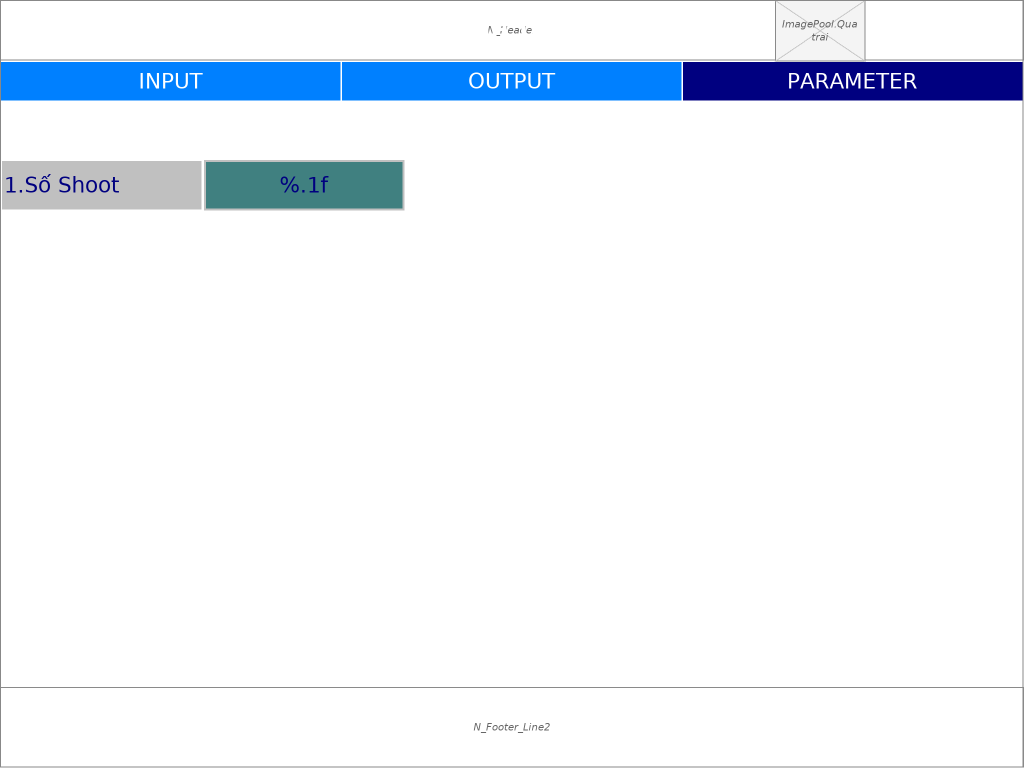
VISUALIZATION N_Parameter_2  // 1024x768
    Frame (0,0 1024x60)
        shows N_Header()
    Rectangle (0,61 341x40), "INPUT"
        OnMouseClick: change screen: N_PLC_I2
    Rectangle (341,61 341x40), "OUTPUT"
        OnMouseClick: change screen: N_PLC_O2
    Rectangle (682,61 341x40), "PARAMETER"
        OnMouseClick: change screen: N_Parameter_2
    Textfield (363,5 400x50), "MÀN HÌNH THÔNG SỐ TRẠM 2"
    Rectangle (1,160 201x50), "1.Số Shoot"
    Textfield (204,160 200x50), "%.1f", text variable: nShoot2
    Image (775,0 90x61), image: ImagePool.Qua trai
        OnMouseClick: change screen: N_Parameter_1
    Frame (0,687 1024x80)
        shows N_Footer_Line2()
END_VISUALIZATION

(* stored: Version 1.1.0.1, ProductVersion 3.1.4024.12
   Visu N_Parameter_2: Id {b5ac443c-cc2c-4eb8-ae59-c64554d53e18} *)
